{attribute 'GeneratedUsingTerminal: KL3361'}
{attribute addProperty BoxType "KL3361"}
{attribute addProperty Id "Channel_1AT %Q*Channel_78571FB40"}
{attribute addProperty CRC "1942717114"}
{attribute addProperty Size "0"}
TYPE KL3361_73CB82BA :
STRUCT
	{attribute addProperty Name "Channel_1"}
	Channel_1 : Channel_78571FB4;
END_STRUCT
END_TYPE

(* stored: Version 1.2.0.0, ProductVersion 3.1.4024.9
   DUT KL3361_73CB82BA: Id {2f757daa-bdbe-48f2-a63f-189384a4e35c} *)
